{attribute 'GeneratedUsingTerminal: EK1122-0000-0018'}
{attribute addProperty BoxType "EK1122-0000-0018"}
{attribute addProperty Id "Beckhoff_ELM9xxxsub_EK1100EK1100_1FC0878B2"}
{attribute addProperty CRC "3361227811"}
{attribute addProperty Size "2"}
TYPE Beckhoff_ELM9xxxEK1122_C8584423 EXTENDS EK1122_1FC0878B :
STRUCT
	{attribute addProperty Name "Beckhoff_ELM9xxxsub_EK1100"}
	{attribute addProperty PreviousPort "Beckhoff ELM9xxxEK1122 : D"}
	Beckhoff_ELM9xxxsub_EK1100 : EK1100_1FC0878B;
END_STRUCT
END_TYPE

(* stored: Version 1.2.0.0, ProductVersion 3.1.4024.9
   DUT Beckhoff_ELM9xxxEK1122_C8584423: Id {9005f2d0-ea74-4330-a0ae-02fa8eebb3bd} *)
